ABB RobotStudio station: material handling 05.03.2024.rsstn

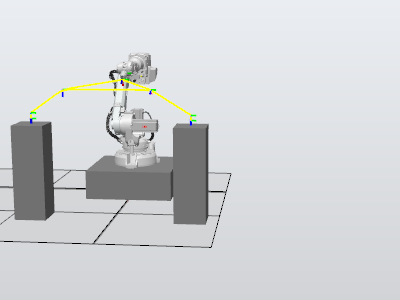
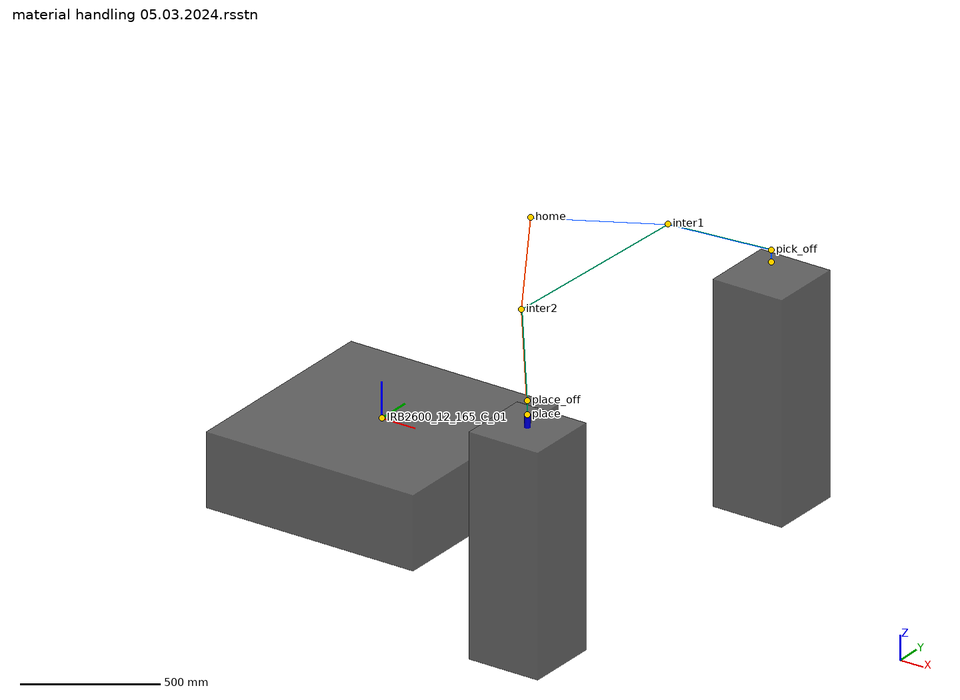
[picture v1: parts stored in the station drawn from their meshes, with robot base, taught points and paths (robot models come from the ABB library and are not in the file)]
Station Station (saved by RobotStudio 22.3.10141.1)
Controller Controller10, task T_ROB1: task frame (RAPID world) sits at (0, 0, 300) mm in the station
Controller Controller10
  mechanical unit ROB_1: IRB2600_12_165_C_01, 6 joints, base frame (0, 0, 0) mm
Layout (positions relative to the parent item):
  - IRB2600_12_165_C_01 [mechanism, from %ABB.RobotStudio.Models.IRB2600%\IRB2600_12_165_C_01.rslib] at (0, 0, 300) mm; joint values [0, -0.7377, 0.7409, 0, 0.5204, 0] (rad or m)
  - Part_1 [part] at (-450, -450, 0) mm, size 900 x 900 x 300 mm
  - SmartComponent_1 [smart component] at (548.16, 0, 1332.96) mm, rotated rx -180 ry 60 rz -180 deg
      signals: DI Attach
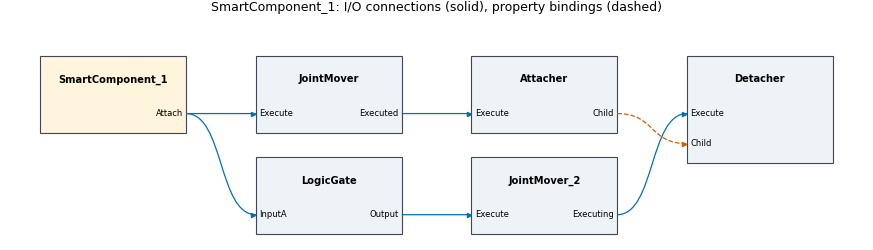
      connections:
        SmartComponent_1.Attach -> JointMover.Execute
        JointMover.Executed -> Attacher.Execute
        SmartComponent_1.Attach -> LogicGate.InputA
        LogicGate.Output -> JointMover_2.Execute
        JointMover_2.Executing -> Detacher.Execute
        Attacher.Child => Detacher.Child
    - Smart_Gripper_Servo_Fingers [mechanism, from Tools\ABB_Smart_Gripper_Servo_Fingers.rslib] at (0, 0, 0) mm; joint values [0.025] (rad or m)
    - Attacher [smart component, from Components\Attacher.rslib]
        properties: Parent=Smart_Gripper_Servo_Fingers; Flange=0; Child=Object; Mount=false; Offset=[0 0 0]; Orientation=[0 0 0]
    - Detacher [smart component, from Components\Detacher.rslib]
        properties: Child=Object; KeepPosition=true
    - JointMover [smart component, from Components\JointMover.rslib]
        properties: Mechanism=Smart_Gripper_Servo_Fingers; Relative=false; Duration=0; J1=0.012
    - LogicGate [smart component, from Components\LogicGate.rslib]
        properties: Operator=NOT; Delay=0
    - JointMover_2 [smart component, from Components\JointMover.rslib]
        properties: Mechanism=Smart_Gripper_Servo_Fingers; Relative=false; Duration=0; J1=0.025
  - Table1 [part] at (1022.32, 593.72, 0) mm, size 300 x 300 x 900 mm
  - Table2 [part] at (1022.32, -921.45, 0) mm, size 300 x 300 x 900 mm
  - Object [part] at (1172.32, -5316.95, 900) mm, size 24 x 23.9 x 50 mm
  - Object_2 [part] at (1172.32, -771.45, 900) mm, size 24 x 23.9 x 50 mm
Attachment: SmartComponent_1 is attached to IRB2600_12_165_C_01 / Link6
Collision set CollisionSet_1:  against , near miss 0 m
Station logic (signal -> signal, property => property):
  Controller10.attach -> SmartComponent_1.Attach
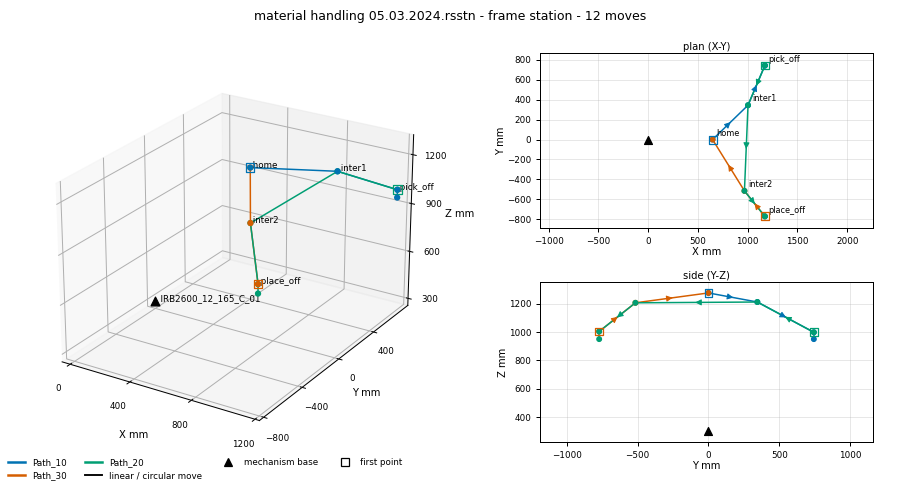
[picture p0: tool path of material handling 05.03.2024.rsstn in frame station, 12 of 12 moves have a stored position in this frame; points joined in program order, loops and branches not executed]
Targets, tools, work objects and paths stored in the station, written as RAPID:
! task T_ROB1
MODULE CalibData
  PERS tooldata Servo:=[TRUE,[[0,0,114.2],[1,0,0,0]],[0.215,[8.7,12.3,49.2],[1,0,0,0],0.00021,0.00024,0.00009]];
ENDMODULE

! task T_ROB1
MODULE Module1
  CONST robtarget home:=[[647.0607775,0,975.863103616],[0.499999994,0,0.866025407,0],[0,0,0,0],[9E+09,9E+09,9E+09,9E+09,9E+09,9E+09]];
  CONST robtarget inter1:=[[1003.205991901,345.00249927,911.778650125],[0.500000008,0.000000009,0.866025399,0.000000014],[0,-1,0,0],[9E+09,9E+09,9E+09,9E+09,9E+09,9E+09]];
  CONST robtarget pick:=[[1172.319028613,743.717020879,650.000245611],[0.014827505,0.044261549,-0.998604866,0.024685666],[0,-1,0,0],[9E+09,9E+09,9E+09,9E+09,9E+09,9E+09]];
  CONST robtarget pick_off:=[[1172.319039553,743.717025339,698.189970311],[0.014827505,0.044261557,-0.998604865,0.024685672],[0,-1,0,0],[9E+09,9E+09,9E+09,9E+09,9E+09,9E+09]];
  CONST robtarget inter2:=[[967.320300012,-515.49547298,906.258010227],[0.014827512,0.044261537,-0.998604868,0.024685618],[-1,-1,-1,0],[9E+09,9E+09,9E+09,9E+09,9E+09,9E+09]];
  CONST robtarget place:=[[1172.319028196,-771.44868311,650.00025774],[0.014827464,0.044261534,-0.998604868,0.024685643],[-1,-1,-1,0],[9E+09,9E+09,9E+09,9E+09,9E+09,9E+09]];
  CONST robtarget place_off:=[[1172.319039404,-771.448687507,703.940245388],[0.014827431,0.044261513,-0.998604869,0.024685658],[-1,-1,-1,0],[9E+09,9E+09,9E+09,9E+09,9E+09,9E+09]];
  PROC Path_10()
    MoveL home,v1000,z100,Servo\WObj:=wobj0;
    MoveL inter1,v1000,z100,Servo\WObj:=wobj0;
    MoveL pick_off,v1000,z100,Servo\WObj:=wobj0;
    MoveL pick,v1000,z100,Servo\WObj:=wobj0;
    WaitTime 1;
    SetDO attach,1;
    WaitTime 1;
  ENDPROC
  PROC Path_30()
    MoveL place_off,v1000,z100,Servo\WObj:=wobj0;
    MoveL inter2,v1000,z100,Servo\WObj:=wobj0;
    MoveL home,v1000,z100,Servo\WObj:=wobj0;
  ENDPROC
  PROC Path_40()
    Path_10;
    Path_20;
    Path_30;
  ENDPROC
  PROC Path_20()
    MoveL pick_off,v1000,z100,Servo\WObj:=wobj0;
    MoveL inter1,v1000,z100,Servo\WObj:=wobj0;
    MoveL inter2,v1000,z100,Servo\WObj:=wobj0;
    MoveL place_off,v1000,z100,Servo\WObj:=wobj0;
    MoveL place,v1000,z100,Servo\WObj:=wobj0;
    WaitTime 1;
    SetDO attach,0;
    WaitTime 1;
  ENDPROC
ENDMODULE

